FUNCTION_BLOCK FB_InvocationControlTestTask EXTENDS TcBase.FB_Task
VAR CONSTANT
    cDefaultCyclesToRun:        UDINT := 1;
END_VAR
VAR
    _nCyclesToRunIn:            UDINT;

    _nCyclesToRun:              UDINT := 10;
    _nCycleCounter:             UDINT;
END_VAR

PROPERTY nCycleCounter : UDINT
GET
nCycleCounter := THIS^._nCycleCounter;
END_GET
END_PROPERTY

METHOD PROTECTED OnStart
VAR_INPUT
END_VAR
IF THIS^._nCyclesToRunIn > 0 THEN
    THIS^._nCyclesToRun := THIS^._nCyclesToRunIn;
ELSE
    THIS^._nCyclesToRun := THIS^.cDefaultCyclesToRun;
END_IF
END_METHOD

METHOD Restore : I_Restorable
Restore := SUPER^.Restore();

THIS^._nCycleCounter := 0;
END_METHOD

METHOD Run : BOOL
VAR_INPUT
END_VAR
IF THIS^.Execute() THEN
    THIS^._nCycleCounter := THIS^._nCycleCounter + 1;

    THIS^.DoneWhen(THIS^._nCycleCounter = THIS^._nCyclesToRun);
END_IF
END_METHOD

METHOD SetRunCondition : REFERENCE TO FB_InvocationControlTestTask
VAR_INPUT
    nCyclesToRun:        UDINT; // Number of cycles to run
END_VAR
SetRunCondition REF= THIS^;

THIS^._nCyclesToRunIn := nCyclesToRun;

THIS^.Invoke();
END_METHOD

END_FUNCTION_BLOCK

(* stored: Version 1.1.0.1, ProductVersion 3.1.4024.12
   POU FB_InvocationControlTestTask: Id {3875f5d6-2f98-4437-917b-772aa7a29e88}, SpecialFunc None
   Property nCycleCounter: Id {00b86a5a-4173-46b2-991f-6722b6a8675b}
   Get Get: Id {8a46db6b-6e56-4661-9681-761cdfc0d7ce}
   Method OnStart: Id {60d6bb11-22ae-499f-a8e5-bc55afadd045}
   Method Restore: Id {50b64149-5c10-46ae-9dda-92f640903083}
   Method Run: Id {a11e5a69-3166-40ec-a4f1-5ca469a7936a}
   Method SetRunCondition: Id {d408fa0c-5788-4b96-999a-24c1be0fb92f} *)
